# EPICS StreamDevice protocol: tests/samples/patterns/mydevice/mydevice.proto
Terminator = CR LF;
getX { out "X?"; in "%f"; }
